// TIA Portal V17 export
// export: Created 2025-06-26T07:49:35.4692747Z, ExportSetting WithDefaults, DisplayName Totally Integrated Automation Portal, DisplayVersion V17 Update 8, DisplayName TIA Portal Openness, DisplayVersion V17 Update 8, DisplayName TIA Portal Version Control Interface, DisplayVersion V17, DisplayName STEP 7 Professional, DisplayVersion V17 Update 8, DisplayName STEP 7 Safety, DisplayVersion V17 Update 6, DisplayName WinCC Advanced, DisplayVersion V17 Update 8
DATA_BLOCK "DB_StaticData"   // DB32
{ S7_Optimized_Access := 'TRUE' }
AUTHOR : AZ
VERSION : 0.1
// stored: AutoNumber true, DBAccessibleFromOPCUA true, DBAccessibleFromWebserver true, InstanceOfName StaticData-STRUCT, InstanceOfType UDT, IsOnlyStoredInLoadMemory true, IsWriteProtectedInAS false
"StaticData-STRUCT"
   // VAR
   //    Fluids { ExternalAccessible := 'False'; ExternalVisible := 'False'; ExternalWritable := 'False'; S7_SetPoint := 'True'} : Array[1..4] of "FluidData-STRUCT";
   //    CompressorTypes { ExternalAccessible := 'False'; ExternalVisible := 'False'; ExternalWritable := 'False'; S7_SetPoint := 'True'} : Array[1..4] of "CompressorData-STRUCT";
   //    SystemTypes { ExternalAccessible := 'False'; ExternalVisible := 'False'; ExternalWritable := 'False'; S7_SetPoint := 'True'} : Array[1..6] of "SystemData-STRUCT";
   // END_VAR
BEGIN
   Fluids[1]."Name" := 'R515B';
   Fluids[2]."Name" := 'R1233zdE';
   Fluids[1].FluidTypeNumber := 1;
   Fluids[2].FluidTypeNumber := 2;
   Fluids[3].FluidTypeNumber := 3;
   Fluids[4].FluidTypeNumber := 4;
   Fluids[1].SaturationCurve_Temperature_C[0] := -43.0;
   Fluids[1].SaturationCurve_Temperature_C[1] := -39.15;
   Fluids[1].SaturationCurve_Temperature_C[2] := -35.31;
   Fluids[1].SaturationCurve_Temperature_C[3] := -31.46;
   Fluids[1].SaturationCurve_Temperature_C[4] := -27.62;
   Fluids[1].SaturationCurve_Temperature_C[5] := -23.77;
   Fluids[1].SaturationCurve_Temperature_C[6] := -19.92;
   Fluids[1].SaturationCurve_Temperature_C[7] := -16.08;
   Fluids[1].SaturationCurve_Temperature_C[8] := -12.23;
   Fluids[1].SaturationCurve_Temperature_C[9] := -8.38;
   Fluids[1].SaturationCurve_Temperature_C[10] := -4.54;
   Fluids[1].SaturationCurve_Temperature_C[11] := -0.69;
   Fluids[1].SaturationCurve_Temperature_C[12] := 3.15;
   Fluids[1].SaturationCurve_Temperature_C[13] := 7.0;
   Fluids[1].SaturationCurve_Temperature_C[14] := 10.85;
   Fluids[1].SaturationCurve_Temperature_C[15] := 14.69;
   Fluids[1].SaturationCurve_Temperature_C[16] := 18.54;
   Fluids[1].SaturationCurve_Temperature_C[17] := 22.38;
   Fluids[1].SaturationCurve_Temperature_C[18] := 26.23;
   Fluids[1].SaturationCurve_Temperature_C[19] := 30.08;
   Fluids[1].SaturationCurve_Temperature_C[20] := 33.92;
   Fluids[1].SaturationCurve_Temperature_C[21] := 37.77;
   Fluids[1].SaturationCurve_Temperature_C[22] := 41.62;
   Fluids[1].SaturationCurve_Temperature_C[23] := 45.46;
   Fluids[1].SaturationCurve_Temperature_C[24] := 49.31;
   Fluids[1].SaturationCurve_Temperature_C[25] := 53.15;
   Fluids[1].SaturationCurve_Temperature_C[26] := 57.0;
   Fluids[1].SaturationCurve_Temperature_C[27] := 60.85;
   Fluids[1].SaturationCurve_Temperature_C[28] := 64.69;
   Fluids[1].SaturationCurve_Temperature_C[29] := 68.54;
   Fluids[1].SaturationCurve_Temperature_C[30] := 72.38;
   Fluids[1].SaturationCurve_Temperature_C[31] := 76.23;
   Fluids[1].SaturationCurve_Temperature_C[32] := 80.08;
   Fluids[1].SaturationCurve_Temperature_C[33] := 83.92;
   Fluids[1].SaturationCurve_Temperature_C[34] := 87.77;
   Fluids[1].SaturationCurve_Temperature_C[35] := 91.62;
   Fluids[1].SaturationCurve_Temperature_C[36] := 95.46;
   Fluids[1].SaturationCurve_Temperature_C[37] := 99.31;
   Fluids[1].SaturationCurve_Temperature_C[38] := 103.15;
   Fluids[1].SaturationCurve_Temperature_C[39] := 107.0;
   Fluids[1].SaturationCurve_Temperature_C[40] := 107.73;
   Fluids[2].SaturationCurve_Temperature_C[0] := -10.0;
   Fluids[2].SaturationCurve_Temperature_C[1] := -5.4872;
   Fluids[2].SaturationCurve_Temperature_C[2] := -0.9744;
   Fluids[2].SaturationCurve_Temperature_C[3] := 3.5385;
   Fluids[2].SaturationCurve_Temperature_C[4] := 8.0513;
   Fluids[2].SaturationCurve_Temperature_C[5] := 12.5641;
   Fluids[2].SaturationCurve_Temperature_C[6] := 17.0769;
   Fluids[2].SaturationCurve_Temperature_C[7] := 21.5897;
   Fluids[2].SaturationCurve_Temperature_C[8] := 26.1026;
   Fluids[2].SaturationCurve_Temperature_C[9] := 30.6154;
   Fluids[2].SaturationCurve_Temperature_C[10] := 35.1282;
   Fluids[2].SaturationCurve_Temperature_C[11] := 39.641;
   Fluids[2].SaturationCurve_Temperature_C[12] := 44.1538;
   Fluids[2].SaturationCurve_Temperature_C[13] := 48.6667;
   Fluids[2].SaturationCurve_Temperature_C[14] := 53.1795;
   Fluids[2].SaturationCurve_Temperature_C[15] := 57.6923;
   Fluids[2].SaturationCurve_Temperature_C[16] := 62.2051;
   Fluids[2].SaturationCurve_Temperature_C[17] := 66.7179;
   Fluids[2].SaturationCurve_Temperature_C[18] := 71.2308;
   Fluids[2].SaturationCurve_Temperature_C[19] := 75.7436;
   Fluids[2].SaturationCurve_Temperature_C[20] := 80.2564;
   Fluids[2].SaturationCurve_Temperature_C[21] := 84.7692;
   Fluids[2].SaturationCurve_Temperature_C[22] := 89.2821;
   Fluids[2].SaturationCurve_Temperature_C[23] := 93.7949;
   Fluids[2].SaturationCurve_Temperature_C[24] := 98.3077;
   Fluids[2].SaturationCurve_Temperature_C[25] := 102.8205;
   Fluids[2].SaturationCurve_Temperature_C[26] := 107.3333;
   Fluids[2].SaturationCurve_Temperature_C[27] := 111.8462;
   Fluids[2].SaturationCurve_Temperature_C[28] := 116.359;
   Fluids[2].SaturationCurve_Temperature_C[29] := 120.8718;
   Fluids[2].SaturationCurve_Temperature_C[30] := 125.3846;
   Fluids[2].SaturationCurve_Temperature_C[31] := 129.8974;
   Fluids[2].SaturationCurve_Temperature_C[32] := 134.4103;
   Fluids[2].SaturationCurve_Temperature_C[33] := 138.9231;
   Fluids[2].SaturationCurve_Temperature_C[34] := 143.4359;
   Fluids[2].SaturationCurve_Temperature_C[35] := 147.9487;
   Fluids[2].SaturationCurve_Temperature_C[36] := 152.4615;
   Fluids[2].SaturationCurve_Temperature_C[37] := 156.9744;
   Fluids[2].SaturationCurve_Temperature_C[38] := 161.4872;
   Fluids[2].SaturationCurve_Temperature_C[39] := 166.0;
   Fluids[2].SaturationCurve_Temperature_C[40] := 172.9092;
   Fluids[1].SaturationCurve_Pressure_kPa[0] := 30.9;
   Fluids[1].SaturationCurve_Pressure_kPa[1] := 38.1;
   Fluids[1].SaturationCurve_Pressure_kPa[2] := 46.5;
   Fluids[1].SaturationCurve_Pressure_kPa[3] := 56.4;
   Fluids[1].SaturationCurve_Pressure_kPa[4] := 67.9;
   Fluids[1].SaturationCurve_Pressure_kPa[5] := 81.1;
   Fluids[1].SaturationCurve_Pressure_kPa[6] := 96.4;
   Fluids[1].SaturationCurve_Pressure_kPa[7] := 113.8;
   Fluids[1].SaturationCurve_Pressure_kPa[8] := 133.6;
   Fluids[1].SaturationCurve_Pressure_kPa[9] := 156.0;
   Fluids[1].SaturationCurve_Pressure_kPa[10] := 181.2;
   Fluids[1].SaturationCurve_Pressure_kPa[11] := 209.5;
   Fluids[1].SaturationCurve_Pressure_kPa[12] := 241.0;
   Fluids[1].SaturationCurve_Pressure_kPa[13] := 276.1;
   Fluids[1].SaturationCurve_Pressure_kPa[14] := 315.0;
   Fluids[1].SaturationCurve_Pressure_kPa[15] := 358.0;
   Fluids[1].SaturationCurve_Pressure_kPa[16] := 405.2;
   Fluids[1].SaturationCurve_Pressure_kPa[17] := 457.1;
   Fluids[1].SaturationCurve_Pressure_kPa[18] := 513.8;
   Fluids[1].SaturationCurve_Pressure_kPa[19] := 575.8;
   Fluids[1].SaturationCurve_Pressure_kPa[20] := 643.2;
   Fluids[1].SaturationCurve_Pressure_kPa[21] := 716.3;
   Fluids[1].SaturationCurve_Pressure_kPa[22] := 795.6;
   Fluids[1].SaturationCurve_Pressure_kPa[23] := 881.2;
   Fluids[1].SaturationCurve_Pressure_kPa[24] := 973.6;
   Fluids[1].SaturationCurve_Pressure_kPa[25] := 1073.1;
   Fluids[1].SaturationCurve_Pressure_kPa[26] := 1180.0;
   Fluids[1].SaturationCurve_Pressure_kPa[27] := 1294.8;
   Fluids[1].SaturationCurve_Pressure_kPa[28] := 1417.7;
   Fluids[1].SaturationCurve_Pressure_kPa[29] := 1549.2;
   Fluids[1].SaturationCurve_Pressure_kPa[30] := 1689.7;
   Fluids[1].SaturationCurve_Pressure_kPa[31] := 1839.6;
   Fluids[1].SaturationCurve_Pressure_kPa[32] := 1999.6;
   Fluids[1].SaturationCurve_Pressure_kPa[33] := 2169.9;
   Fluids[1].SaturationCurve_Pressure_kPa[34] := 2351.3;
   Fluids[1].SaturationCurve_Pressure_kPa[35] := 2544.5;
   Fluids[1].SaturationCurve_Pressure_kPa[36] := 2750.1;
   Fluids[1].SaturationCurve_Pressure_kPa[37] := 2969.2;
   Fluids[1].SaturationCurve_Pressure_kPa[38] := 3202.9;
   Fluids[1].SaturationCurve_Pressure_kPa[39] := 3453.4;
   Fluids[1].SaturationCurve_Pressure_kPa[40] := 3501.0;
   Fluids[2].SaturationCurve_Pressure_kPa[0] := 30.3567;
   Fluids[2].SaturationCurve_Pressure_kPa[1] := 37.5596;
   Fluids[2].SaturationCurve_Pressure_kPa[2] := 46.0817;
   Fluids[2].SaturationCurve_Pressure_kPa[3] := 56.0903;
   Fluids[2].SaturationCurve_Pressure_kPa[4] := 67.7633;
   Fluids[2].SaturationCurve_Pressure_kPa[5] := 81.2888;
   Fluids[2].SaturationCurve_Pressure_kPa[6] := 96.865;
   Fluids[2].SaturationCurve_Pressure_kPa[7] := 114.6997;
   Fluids[2].SaturationCurve_Pressure_kPa[8] := 135.0095;
   Fluids[2].SaturationCurve_Pressure_kPa[9] := 158.0203;
   Fluids[2].SaturationCurve_Pressure_kPa[10] := 183.9659;
   Fluids[2].SaturationCurve_Pressure_kPa[11] := 213.0886;
   Fluids[2].SaturationCurve_Pressure_kPa[12] := 245.6381;
   Fluids[2].SaturationCurve_Pressure_kPa[13] := 281.8717;
   Fluids[2].SaturationCurve_Pressure_kPa[14] := 322.0539;
   Fluids[2].SaturationCurve_Pressure_kPa[15] := 366.4563;
   Fluids[2].SaturationCurve_Pressure_kPa[16] := 415.3576;
   Fluids[2].SaturationCurve_Pressure_kPa[17] := 469.0435;
   Fluids[2].SaturationCurve_Pressure_kPa[18] := 527.8071;
   Fluids[2].SaturationCurve_Pressure_kPa[19] := 591.9489;
   Fluids[2].SaturationCurve_Pressure_kPa[20] := 661.7775;
   Fluids[2].SaturationCurve_Pressure_kPa[21] := 737.6098;
   Fluids[2].SaturationCurve_Pressure_kPa[22] := 819.7723;
   Fluids[2].SaturationCurve_Pressure_kPa[23] := 908.6015;
   Fluids[2].SaturationCurve_Pressure_kPa[24] := 1004.446;
   Fluids[2].SaturationCurve_Pressure_kPa[25] := 1107.666;
   Fluids[2].SaturationCurve_Pressure_kPa[26] := 1218.639;
   Fluids[2].SaturationCurve_Pressure_kPa[27] := 1337.757;
   Fluids[2].SaturationCurve_Pressure_kPa[28] := 1465.436;
   Fluids[2].SaturationCurve_Pressure_kPa[29] := 1602.111;
   Fluids[2].SaturationCurve_Pressure_kPa[30] := 1748.251;
   Fluids[2].SaturationCurve_Pressure_kPa[31] := 1904.356;
   Fluids[2].SaturationCurve_Pressure_kPa[32] := 2070.969;
   Fluids[2].SaturationCurve_Pressure_kPa[33] := 2248.688;
   Fluids[2].SaturationCurve_Pressure_kPa[34] := 2438.177;
   Fluids[2].SaturationCurve_Pressure_kPa[35] := 2640.193;
   Fluids[2].SaturationCurve_Pressure_kPa[36] := 2855.623;
   Fluids[2].SaturationCurve_Pressure_kPa[37] := 3085.555;
   Fluids[2].SaturationCurve_Pressure_kPa[38] := 3331.466;
   Fluids[2].SaturationCurve_Pressure_kPa[39] := 3595.998;
   Fluids[2].SaturationCurve_Pressure_kPa[40] := 4001.0;
   Fluids[1].DensityCurve_Pressure_kPa[0] := 50.0;
   Fluids[1].DensityCurve_Pressure_kPa[1] := 100.0;
   Fluids[1].DensityCurve_Pressure_kPa[2] := 220.0;
   Fluids[1].DensityCurve_Pressure_kPa[3] := 390.0;
   Fluids[1].DensityCurve_Pressure_kPa[4] := 600.0;
   Fluids[1].DensityCurve_Pressure_kPa[5] := 850.0;
   Fluids[1].DensityCurve_Pressure_kPa[6] := 1200.0;
   Fluids[1].DensityCurve_Pressure_kPa[7] := 1500.0;
   Fluids[1].DensityCurve_Pressure_kPa[8] := 1900.0;
   Fluids[1].DensityCurve_Pressure_kPa[9] := 2400.0;
   Fluids[1].DensityCurve_Pressure_kPa[10] := 2900.0;
   Fluids[1].DensityCurve_Pressure_kPa[11] := 3400.0;
   Fluids[1].DensityCurve_Pressure_kPa[12] := 4000.0;
   Fluids[2].DensityCurve_Pressure_kPa[0] := 50.0;
   Fluids[2].DensityCurve_Pressure_kPa[1] := 74.7475;
   Fluids[2].DensityCurve_Pressure_kPa[2] := 173.05;
   Fluids[2].DensityCurve_Pressure_kPa[3] := 388.0866;
   Fluids[2].DensityCurve_Pressure_kPa[4] := 746.4811;
   Fluids[2].DensityCurve_Pressure_kPa[5] := 1244.251;
   Fluids[2].DensityCurve_Pressure_kPa[6] := 1836.598;
   Fluids[2].DensityCurve_Pressure_kPa[7] := 2441.284;
   Fluids[2].DensityCurve_Pressure_kPa[8] := 2962.33;
   Fluids[2].DensityCurve_Pressure_kPa[9] := 3328.69;
   Fluids[2].DensityCurve_Pressure_kPa[10] := 3526.57;
   Fluids[2].DensityCurve_Pressure_kPa[11] := 3613.637;
   Fluids[2].DensityCurve_Pressure_kPa[12] := 4001.0;
   Fluids[1].DensityCurveLiquide_Densety_kg_m3[0] := 1354.6;
   Fluids[1].DensityCurveLiquide_Densety_kg_m3[1] := 1314.3;
   Fluids[1].DensityCurveLiquide_Densety_kg_m3[2] := 1257.6;
   Fluids[1].DensityCurveLiquide_Densety_kg_m3[3] := 1206.1;
   Fluids[1].DensityCurveLiquide_Densety_kg_m3[4] := 1158.8;
   Fluids[1].DensityCurveLiquide_Densety_kg_m3[5] := 1113.0;
   Fluids[1].DensityCurveLiquide_Densety_kg_m3[6] := 1057.8;
   Fluids[1].DensityCurveLiquide_Densety_kg_m3[7] := 1014.5;
   Fluids[1].DensityCurveLiquide_Densety_kg_m3[8] := 958.8;
   Fluids[1].DensityCurveLiquide_Densety_kg_m3[9] := 887.4;
   Fluids[1].DensityCurveLiquide_Densety_kg_m3[10] := 805.7;
   Fluids[1].DensityCurveLiquide_Densety_kg_m3[11] := 685.3;
   Fluids[1].DensityCurveLiquide_Densety_kg_m3[12] := 761.3;
   Fluids[2].DensityCurveLiquide_Densety_kg_m3[0] := 1319.278;
   Fluids[2].DensityCurveLiquide_Densety_kg_m3[1] := 1297.254;
   Fluids[2].DensityCurveLiquide_Densety_kg_m3[2] := 1242.459;
   Fluids[2].DensityCurveLiquide_Densety_kg_m3[3] := 1173.489;
   Fluids[2].DensityCurveLiquide_Densety_kg_m3[4] := 1098.545;
   Fluids[2].DensityCurveLiquide_Densety_kg_m3[5] := 1019.4;
   Fluids[2].DensityCurveLiquide_Densety_kg_m3[6] := 936.68;
   Fluids[2].DensityCurveLiquide_Densety_kg_m3[7] := 851.4562;
   Fluids[2].DensityCurveLiquide_Densety_kg_m3[8] := 765.7374;
   Fluids[2].DensityCurveLiquide_Densety_kg_m3[9] := 682.3312;
   Fluids[2].DensityCurveLiquide_Densety_kg_m3[10] := 605.4245;
   Fluids[2].DensityCurveLiquide_Densety_kg_m3[11] := 523.5075;
   Fluids[2].DensityCurveLiquide_Densety_kg_m3[12] := 455.9911;
   Fluids[1].DensityCurveVapor_Densety_kg_m3[0] := 3.03;
   Fluids[1].DensityCurveVapor_Densety_kg_m3[1] := 5.8;
   Fluids[1].DensityCurveVapor_Densety_kg_m3[2] := 12.25;
   Fluids[1].DensityCurveVapor_Densety_kg_m3[3] := 21.3;
   Fluids[1].DensityCurveVapor_Densety_kg_m3[4] := 32.65;
   Fluids[1].DensityCurveVapor_Densety_kg_m3[5] := 46.66;
   Fluids[1].DensityCurveVapor_Densety_kg_m3[6] := 67.55;
   Fluids[1].DensityCurveVapor_Densety_kg_m3[7] := 87.0;
   Fluids[1].DensityCurveVapor_Densety_kg_m3[8] := 115.92;
   Fluids[1].DensityCurveVapor_Densety_kg_m3[9] := 159.17;
   Fluids[1].DensityCurveVapor_Densety_kg_m3[10] := 216.59;
   Fluids[1].DensityCurveVapor_Densety_kg_m3[11] := 315.0;
   Fluids[1].DensityCurveVapor_Densety_kg_m3[12] := 761.33;
   Fluids[2].DensityCurveVapor_Densety_kg_m3[0] := 2.9405;
   Fluids[2].DensityCurveVapor_Densety_kg_m3[1] := 4.2862;
   Fluids[2].DensityCurveVapor_Densety_kg_m3[2] := 9.4624;
   Fluids[2].DensityCurveVapor_Densety_kg_m3[3] := 20.5809;
   Fluids[2].DensityCurveVapor_Densety_kg_m3[4] := 39.5976;
   Fluids[2].DensityCurveVapor_Densety_kg_m3[5] := 68.316;
   Fluids[2].DensityCurveVapor_Densety_kg_m3[6] := 108.1358;
   Fluids[2].DensityCurveVapor_Densety_kg_m3[7] := 159.5525;
   Fluids[2].DensityCurveVapor_Densety_kg_m3[8] := 221.352;
   Fluids[2].DensityCurveVapor_Densety_kg_m3[9] := 289.9457;
   Fluids[2].DensityCurveVapor_Densety_kg_m3[10] := 359.0497;
   Fluids[2].DensityCurveVapor_Densety_kg_m3[11] := 437.3655;
   Fluids[2].DensityCurveVapor_Densety_kg_m3[12] := 455.9911;
   Fluids[1].DensityCurveVapor_SuperheatCorrection_a := 1.3561E-07;
   Fluids[2].DensityCurveVapor_SuperheatCorrection_a := 0.0;
   Fluids[1].DensityCurveVapor_SuperheatCorrection_b := 0.00019589;
   Fluids[2].DensityCurveVapor_SuperheatCorrection_b := 0.0002;
   Fluids[1].EnthalpyMap_Superheat_C[0] := -20.0;
   Fluids[1].EnthalpyMap_Superheat_C[1] := -6.0;
   Fluids[1].EnthalpyMap_Superheat_C[2] := -2.0;
   Fluids[1].EnthalpyMap_Superheat_C[3] := -0.01;
   Fluids[1].EnthalpyMap_Superheat_C[4] := 0.01;
   Fluids[1].EnthalpyMap_Superheat_C[5] := 2.0;
   Fluids[1].EnthalpyMap_Superheat_C[6] := 6.0;
   Fluids[1].EnthalpyMap_Superheat_C[7] := 18.0;
   Fluids[1].EnthalpyMap_Superheat_C[8] := 40.0;
   Fluids[2].EnthalpyMap_Superheat_C[0] := -20.0;
   Fluids[2].EnthalpyMap_Superheat_C[1] := -6.0;
   Fluids[2].EnthalpyMap_Superheat_C[2] := -2.0;
   Fluids[2].EnthalpyMap_Superheat_C[3] := -0.01;
   Fluids[2].EnthalpyMap_Superheat_C[4] := 0.01;
   Fluids[2].EnthalpyMap_Superheat_C[5] := 2.0;
   Fluids[2].EnthalpyMap_Superheat_C[6] := 6.0;
   Fluids[2].EnthalpyMap_Superheat_C[7] := 18.0;
   Fluids[2].EnthalpyMap_Superheat_C[8] := 40.0;
   Fluids[1].EnthalpyMap_Pressure_kPa[0] := 100.0;
   Fluids[1].EnthalpyMap_Pressure_kPa[1] := 220.0;
   Fluids[1].EnthalpyMap_Pressure_kPa[2] := 390.0;
   Fluids[1].EnthalpyMap_Pressure_kPa[3] := 600.0;
   Fluids[1].EnthalpyMap_Pressure_kPa[4] := 850.0;
   Fluids[1].EnthalpyMap_Pressure_kPa[5] := 1200.0;
   Fluids[1].EnthalpyMap_Pressure_kPa[6] := 1500.0;
   Fluids[1].EnthalpyMap_Pressure_kPa[7] := 1900.0;
   Fluids[1].EnthalpyMap_Pressure_kPa[8] := 2400.0;
   Fluids[1].EnthalpyMap_Pressure_kPa[9] := 2900.0;
   Fluids[1].EnthalpyMap_Pressure_kPa[10] := 3400.0;
   Fluids[1].EnthalpyMap_Pressure_kPa[11] := 4000.0;
   Fluids[2].EnthalpyMap_Pressure_kPa[0] := 100.0;
   Fluids[2].EnthalpyMap_Pressure_kPa[1] := 127.0833;
   Fluids[2].EnthalpyMap_Pressure_kPa[2] := 234.6644;
   Fluids[2].EnthalpyMap_Pressure_kPa[3] := 469.9978;
   Fluids[2].EnthalpyMap_Pressure_kPa[4] := 862.2203;
   Fluids[2].EnthalpyMap_Pressure_kPa[5] := 1406.974;
   Fluids[2].EnthalpyMap_Pressure_kPa[6] := 2055.23;
   Fluids[2].EnthalpyMap_Pressure_kPa[7] := 2716.992;
   Fluids[2].EnthalpyMap_Pressure_kPa[8] := 3287.218;
   Fluids[2].EnthalpyMap_Pressure_kPa[9] := 3688.158;
   Fluids[2].EnthalpyMap_Pressure_kPa[10] := 3904.715;
   Fluids[2].EnthalpyMap_Pressure_kPa[11] := 4000.0;
   Fluids[1].EnthalpyMap_Enthalpy_kJ_kg[0,0] := 150.5;
   Fluids[1].EnthalpyMap_Enthalpy_kJ_kg[0,1] := 167.9;
   Fluids[1].EnthalpyMap_Enthalpy_kJ_kg[0,2] := 173.0;
   Fluids[1].EnthalpyMap_Enthalpy_kJ_kg[0,3] := 175.5;
   Fluids[1].EnthalpyMap_Enthalpy_kJ_kg[0,4] := 271.8;
   Fluids[1].EnthalpyMap_Enthalpy_kJ_kg[0,5] := 367.3;
   Fluids[1].EnthalpyMap_Enthalpy_kJ_kg[0,6] := 370.6;
   Fluids[1].EnthalpyMap_Enthalpy_kJ_kg[0,7] := 380.6;
   Fluids[1].EnthalpyMap_Enthalpy_kJ_kg[0,8] := 399.6;
   Fluids[1].EnthalpyMap_Enthalpy_kJ_kg[1,0] := 175.2;
   Fluids[1].EnthalpyMap_Enthalpy_kJ_kg[1,1] := 193.0;
   Fluids[1].EnthalpyMap_Enthalpy_kJ_kg[1,2] := 198.2;
   Fluids[1].EnthalpyMap_Enthalpy_kJ_kg[1,3] := 200.8;
   Fluids[1].EnthalpyMap_Enthalpy_kJ_kg[1,4] := 297.6;
   Fluids[1].EnthalpyMap_Enthalpy_kJ_kg[1,5] := 381.1;
   Fluids[1].EnthalpyMap_Enthalpy_kJ_kg[1,6] := 384.6;
   Fluids[1].EnthalpyMap_Enthalpy_kJ_kg[1,7] := 395.3;
   Fluids[1].EnthalpyMap_Enthalpy_kJ_kg[1,8] := 415.2;
   Fluids[1].EnthalpyMap_Enthalpy_kJ_kg[2,0] := 196.6;
   Fluids[1].EnthalpyMap_Enthalpy_kJ_kg[2,1] := 214.9;
   Fluids[1].EnthalpyMap_Enthalpy_kJ_kg[2,2] := 220.2;
   Fluids[1].EnthalpyMap_Enthalpy_kJ_kg[2,3] := 222.9;
   Fluids[1].EnthalpyMap_Enthalpy_kJ_kg[2,4] := 318.7;
   Fluids[1].EnthalpyMap_Enthalpy_kJ_kg[2,5] := 392.3;
   Fluids[1].EnthalpyMap_Enthalpy_kJ_kg[2,6] := 396.1;
   Fluids[1].EnthalpyMap_Enthalpy_kJ_kg[2,7] := 407.4;
   Fluids[1].EnthalpyMap_Enthalpy_kJ_kg[2,8] := 428.3;
   Fluids[1].EnthalpyMap_Enthalpy_kJ_kg[3,0] := 215.2;
   Fluids[1].EnthalpyMap_Enthalpy_kJ_kg[3,1] := 234.0;
   Fluids[1].EnthalpyMap_Enthalpy_kJ_kg[3,2] := 239.5;
   Fluids[1].EnthalpyMap_Enthalpy_kJ_kg[3,3] := 242.3;
   Fluids[1].EnthalpyMap_Enthalpy_kJ_kg[3,4] := 336.5;
   Fluids[1].EnthalpyMap_Enthalpy_kJ_kg[3,5] := 401.4;
   Fluids[1].EnthalpyMap_Enthalpy_kJ_kg[3,6] := 405.3;
   Fluids[1].EnthalpyMap_Enthalpy_kJ_kg[3,7] := 417.3;
   Fluids[1].EnthalpyMap_Enthalpy_kJ_kg[3,8] := 439.2;
   Fluids[1].EnthalpyMap_Enthalpy_kJ_kg[4,0] := 232.1;
   Fluids[1].EnthalpyMap_Enthalpy_kJ_kg[4,1] := 251.5;
   Fluids[1].EnthalpyMap_Enthalpy_kJ_kg[4,2] := 257.2;
   Fluids[1].EnthalpyMap_Enthalpy_kJ_kg[4,3] := 260.1;
   Fluids[1].EnthalpyMap_Enthalpy_kJ_kg[4,4] := 352.6;
   Fluids[1].EnthalpyMap_Enthalpy_kJ_kg[4,5] := 408.9;
   Fluids[1].EnthalpyMap_Enthalpy_kJ_kg[4,6] := 413.1;
   Fluids[1].EnthalpyMap_Enthalpy_kJ_kg[4,7] := 425.7;
   Fluids[1].EnthalpyMap_Enthalpy_kJ_kg[4,8] := 448.6;
   Fluids[1].EnthalpyMap_Enthalpy_kJ_kg[5,0] := 251.0;
   Fluids[1].EnthalpyMap_Enthalpy_kJ_kg[5,1] := 271.1;
   Fluids[1].EnthalpyMap_Enthalpy_kJ_kg[5,2] := 277.1;
   Fluids[1].EnthalpyMap_Enthalpy_kJ_kg[5,3] := 280.1;
   Fluids[1].EnthalpyMap_Enthalpy_kJ_kg[5,4] := 370.8;
   Fluids[1].EnthalpyMap_Enthalpy_kJ_kg[5,5] := 416.2;
   Fluids[1].EnthalpyMap_Enthalpy_kJ_kg[5,6] := 420.8;
   Fluids[1].EnthalpyMap_Enthalpy_kJ_kg[5,7] := 434.3;
   Fluids[1].EnthalpyMap_Enthalpy_kJ_kg[5,8] := 458.5;
   Fluids[1].EnthalpyMap_Enthalpy_kJ_kg[6,0] := 264.4;
   Fluids[1].EnthalpyMap_Enthalpy_kJ_kg[6,1] := 285.3;
   Fluids[1].EnthalpyMap_Enthalpy_kJ_kg[6,2] := 291.5;
   Fluids[1].EnthalpyMap_Enthalpy_kJ_kg[6,3] := 294.7;
   Fluids[1].EnthalpyMap_Enthalpy_kJ_kg[6,4] := 384.4;
   Fluids[1].EnthalpyMap_Enthalpy_kJ_kg[6,5] := 420.5;
   Fluids[1].EnthalpyMap_Enthalpy_kJ_kg[6,6] := 425.5;
   Fluids[1].EnthalpyMap_Enthalpy_kJ_kg[6,7] := 439.9;
   Fluids[1].EnthalpyMap_Enthalpy_kJ_kg[6,8] := 465.0;
   Fluids[1].EnthalpyMap_Enthalpy_kJ_kg[7,0] := 279.9;
   Fluids[1].EnthalpyMap_Enthalpy_kJ_kg[7,1] := 301.7;
   Fluids[1].EnthalpyMap_Enthalpy_kJ_kg[7,2] := 308.4;
   Fluids[1].EnthalpyMap_Enthalpy_kJ_kg[7,3] := 311.8;
   Fluids[1].EnthalpyMap_Enthalpy_kJ_kg[7,4] := 401.2;
   Fluids[1].EnthalpyMap_Enthalpy_kJ_kg[7,5] := 424.5;
   Fluids[1].EnthalpyMap_Enthalpy_kJ_kg[7,6] := 430.0;
   Fluids[1].EnthalpyMap_Enthalpy_kJ_kg[7,7] := 445.6;
   Fluids[1].EnthalpyMap_Enthalpy_kJ_kg[7,8] := 472.1;
   Fluids[1].EnthalpyMap_Enthalpy_kJ_kg[8,0] := 296.6;
   Fluids[1].EnthalpyMap_Enthalpy_kJ_kg[8,1] := 319.8;
   Fluids[1].EnthalpyMap_Enthalpy_kJ_kg[8,2] := 327.2;
   Fluids[1].EnthalpyMap_Enthalpy_kJ_kg[8,3] := 331.1;
   Fluids[1].EnthalpyMap_Enthalpy_kJ_kg[8,4] := 422.0;
   Fluids[1].EnthalpyMap_Enthalpy_kJ_kg[8,5] := 427.0;
   Fluids[1].EnthalpyMap_Enthalpy_kJ_kg[8,6] := 433.5;
   Fluids[1].EnthalpyMap_Enthalpy_kJ_kg[8,7] := 450.9;
   Fluids[1].EnthalpyMap_Enthalpy_kJ_kg[8,8] := 479.1;
   Fluids[1].EnthalpyMap_Enthalpy_kJ_kg[9,0] := 311.2;
   Fluids[1].EnthalpyMap_Enthalpy_kJ_kg[9,1] := 336.2;
   Fluids[1].EnthalpyMap_Enthalpy_kJ_kg[9,2] := 344.7;
   Fluids[1].EnthalpyMap_Enthalpy_kJ_kg[9,3] := 349.5;
   Fluids[1].EnthalpyMap_Enthalpy_kJ_kg[9,4] := 421.8;
   Fluids[1].EnthalpyMap_Enthalpy_kJ_kg[9,5] := 426.9;
   Fluids[1].EnthalpyMap_Enthalpy_kJ_kg[9,6] := 435.1;
   Fluids[1].EnthalpyMap_Enthalpy_kJ_kg[9,7] := 454.7;
   Fluids[1].EnthalpyMap_Enthalpy_kJ_kg[9,8] := 484.7;
   Fluids[1].EnthalpyMap_Enthalpy_kJ_kg[10,0] := 324.2;
   Fluids[1].EnthalpyMap_Enthalpy_kJ_kg[10,1] := 351.3;
   Fluids[1].EnthalpyMap_Enthalpy_kJ_kg[10,2] := 361.9;
   Fluids[1].EnthalpyMap_Enthalpy_kJ_kg[10,3] := 370.2;
   Fluids[1].EnthalpyMap_Enthalpy_kJ_kg[10,4] := 413.6;
   Fluids[1].EnthalpyMap_Enthalpy_kJ_kg[10,5] := 423.8;
   Fluids[1].EnthalpyMap_Enthalpy_kJ_kg[10,6] := 434.9;
   Fluids[1].EnthalpyMap_Enthalpy_kJ_kg[10,7] := 457.3;
   Fluids[1].EnthalpyMap_Enthalpy_kJ_kg[10,8] := 489.2;
   Fluids[1].EnthalpyMap_Enthalpy_kJ_kg[11,0] := 339.4;
   Fluids[1].EnthalpyMap_Enthalpy_kJ_kg[11,1] := 370.1;
   Fluids[1].EnthalpyMap_Enthalpy_kJ_kg[11,2] := 387.3;
   Fluids[1].EnthalpyMap_Enthalpy_kJ_kg[11,3] := 407.7;
   Fluids[1].EnthalpyMap_Enthalpy_kJ_kg[11,4] := 407.9;
   Fluids[1].EnthalpyMap_Enthalpy_kJ_kg[11,5] := 421.3;
   Fluids[1].EnthalpyMap_Enthalpy_kJ_kg[11,6] := 435.4;
   Fluids[1].EnthalpyMap_Enthalpy_kJ_kg[11,7] := 460.7;
   Fluids[1].EnthalpyMap_Enthalpy_kJ_kg[11,8] := 494.6;
   Fluids[2].EnthalpyMap_Enthalpy_kJ_kg[0,0] := 197.5698;
   Fluids[2].EnthalpyMap_Enthalpy_kJ_kg[0,1] := 214.1515;
   Fluids[2].EnthalpyMap_Enthalpy_kJ_kg[0,2] := 218.9438;
   Fluids[2].EnthalpyMap_Enthalpy_kJ_kg[0,3] := 221.3373;
   Fluids[2].EnthalpyMap_Enthalpy_kJ_kg[0,4] := 416.1527;
   Fluids[2].EnthalpyMap_Enthalpy_kJ_kg[0,5] := 417.767;
   Fluids[2].EnthalpyMap_Enthalpy_kJ_kg[0,6] := 421.028;
   Fluids[2].EnthalpyMap_Enthalpy_kJ_kg[0,7] := 430.9391;
   Fluids[2].EnthalpyMap_Enthalpy_kJ_kg[0,8] := 449.5907;
   Fluids[2].EnthalpyMap_Enthalpy_kJ_kg[1,0] := 205.2355;
   Fluids[2].EnthalpyMap_Enthalpy_kJ_kg[1,1] := 221.9542;
   Fluids[2].EnthalpyMap_Enthalpy_kJ_kg[1,2] := 226.7875;
   Fluids[2].EnthalpyMap_Enthalpy_kJ_kg[1,3] := 229.2018;
   Fluids[2].EnthalpyMap_Enthalpy_kJ_kg[1,4] := 420.6821;
   Fluids[2].EnthalpyMap_Enthalpy_kJ_kg[1,5] := 422.3276;
   Fluids[2].EnthalpyMap_Enthalpy_kJ_kg[1,6] := 425.6502;
   Fluids[2].EnthalpyMap_Enthalpy_kJ_kg[1,7] := 435.7365;
   Fluids[2].EnthalpyMap_Enthalpy_kJ_kg[1,8] := 454.6786;
   Fluids[2].EnthalpyMap_Enthalpy_kJ_kg[2,0] := 227.161;
   Fluids[2].EnthalpyMap_Enthalpy_kJ_kg[2,1] := 244.2909;
   Fluids[2].EnthalpyMap_Enthalpy_kJ_kg[2,2] := 249.2492;
   Fluids[2].EnthalpyMap_Enthalpy_kJ_kg[2,3] := 251.7272;
   Fluids[2].EnthalpyMap_Enthalpy_kJ_kg[2,4] := 433.2917;
   Fluids[2].EnthalpyMap_Enthalpy_kJ_kg[2,5] := 435.0327;
   Fluids[2].EnthalpyMap_Enthalpy_kJ_kg[2,6] := 438.5429;
   Fluids[2].EnthalpyMap_Enthalpy_kJ_kg[2,7] := 449.1592;
   Fluids[2].EnthalpyMap_Enthalpy_kJ_kg[2,8] := 468.9681;
   Fluids[2].EnthalpyMap_Enthalpy_kJ_kg[3,0] := 256.9384;
   Fluids[2].EnthalpyMap_Enthalpy_kJ_kg[3,1] := 274.7034;
   Fluids[2].EnthalpyMap_Enthalpy_kJ_kg[3,2] := 279.8614;
   Fluids[2].EnthalpyMap_Enthalpy_kJ_kg[3,3] := 282.4424;
   Fluids[2].EnthalpyMap_Enthalpy_kJ_kg[3,4] := 449.3674;
   Fluids[2].EnthalpyMap_Enthalpy_kJ_kg[3,5] := 451.2598;
   Fluids[2].EnthalpyMap_Enthalpy_kJ_kg[3,6] := 455.0643;
   Fluids[2].EnthalpyMap_Enthalpy_kJ_kg[3,7] := 466.4958;
   Fluids[2].EnthalpyMap_Enthalpy_kJ_kg[3,8] := 487.595;
   Fluids[2].EnthalpyMap_Enthalpy_kJ_kg[4,0] := 288.6115;
   Fluids[2].EnthalpyMap_Enthalpy_kJ_kg[4,1] := 307.2277;
   Fluids[2].EnthalpyMap_Enthalpy_kJ_kg[4,2] := 312.6681;
   Fluids[2].EnthalpyMap_Enthalpy_kJ_kg[4,3] := 315.398;
   Fluids[2].EnthalpyMap_Enthalpy_kJ_kg[4,4] := 464.6608;
   Fluids[2].EnthalpyMap_Enthalpy_kJ_kg[4,5] := 466.762;
   Fluids[2].EnthalpyMap_Enthalpy_kJ_kg[4,6] := 470.9658;
   Fluids[2].EnthalpyMap_Enthalpy_kJ_kg[4,7] := 483.4603;
   Fluids[2].EnthalpyMap_Enthalpy_kJ_kg[4,8] := 506.1447;
   Fluids[2].EnthalpyMap_Enthalpy_kJ_kg[5,0] := 319.2484;
   Fluids[2].EnthalpyMap_Enthalpy_kJ_kg[5,1] := 339.0134;
   Fluids[2].EnthalpyMap_Enthalpy_kJ_kg[5,2] := 344.8686;
   Fluids[2].EnthalpyMap_Enthalpy_kJ_kg[5,3] := 347.8254;
   Fluids[2].EnthalpyMap_Enthalpy_kJ_kg[5,4] := 476.8875;
   Fluids[2].EnthalpyMap_Enthalpy_kJ_kg[5,5] := 479.2968;
   Fluids[2].EnthalpyMap_Enthalpy_kJ_kg[5,6] := 484.0675;
   Fluids[2].EnthalpyMap_Enthalpy_kJ_kg[5,7] := 497.9603;
   Fluids[2].EnthalpyMap_Enthalpy_kJ_kg[5,8] := 522.524;
   Fluids[2].EnthalpyMap_Enthalpy_kJ_kg[6,0] := 346.9259;
   Fluids[2].EnthalpyMap_Enthalpy_kJ_kg[6,1] := 368.272;
   Fluids[2].EnthalpyMap_Enthalpy_kJ_kg[6,2] := 374.7868;
   Fluids[2].EnthalpyMap_Enthalpy_kJ_kg[6,3] := 378.132;
   Fluids[2].EnthalpyMap_Enthalpy_kJ_kg[6,4] := 484.4899;
   Fluids[2].EnthalpyMap_Enthalpy_kJ_kg[6,5] := 487.4372;
   Fluids[2].EnthalpyMap_Enthalpy_kJ_kg[6,6] := 493.119;
   Fluids[2].EnthalpyMap_Enthalpy_kJ_kg[6,7] := 508.9522;
   Fluids[2].EnthalpyMap_Enthalpy_kJ_kg[6,8] := 535.7144;
   Fluids[2].EnthalpyMap_Enthalpy_kJ_kg[7,0] := 369.9632;
   Fluids[2].EnthalpyMap_Enthalpy_kJ_kg[7,1] := 393.4236;
   Fluids[2].EnthalpyMap_Enthalpy_kJ_kg[7,2] := 401.0829;
   Fluids[2].EnthalpyMap_Enthalpy_kJ_kg[7,3] := 405.235;
   Fluids[2].EnthalpyMap_Enthalpy_kJ_kg[7,4] := 486.2374;
   Fluids[2].EnthalpyMap_Enthalpy_kJ_kg[7,5] := 490.3629;
   Fluids[2].EnthalpyMap_Enthalpy_kJ_kg[7,6] := 497.6848;
   Fluids[2].EnthalpyMap_Enthalpy_kJ_kg[7,7] := 516.2058;
   Fluids[2].EnthalpyMap_Enthalpy_kJ_kg[7,8] := 545.3667;
   Fluids[2].EnthalpyMap_Enthalpy_kJ_kg[8,0] := 387.0381;
   Fluids[2].EnthalpyMap_Enthalpy_kJ_kg[8,1] := 412.9451;
   Fluids[2].EnthalpyMap_Enthalpy_kJ_kg[8,2] := 422.6469;
   Fluids[2].EnthalpyMap_Enthalpy_kJ_kg[8,3] := 429.1883;
   Fluids[2].EnthalpyMap_Enthalpy_kJ_kg[8,4] := 480.7851;
   Fluids[2].EnthalpyMap_Enthalpy_kJ_kg[8,5] := 488.3624;
   Fluids[2].EnthalpyMap_Enthalpy_kJ_kg[8,6] := 498.5881;
   Fluids[2].EnthalpyMap_Enthalpy_kJ_kg[8,7] := 520.3678;
   Fluids[2].EnthalpyMap_Enthalpy_kJ_kg[8,8] := 551.7377;
   Fluids[2].EnthalpyMap_Enthalpy_kJ_kg[9,0] := 397.8677;
   Fluids[2].EnthalpyMap_Enthalpy_kJ_kg[9,1] := 425.8558;
   Fluids[2].EnthalpyMap_Enthalpy_kJ_kg[9,2] := 438.3909;
   Fluids[2].EnthalpyMap_Enthalpy_kJ_kg[9,3] := 462.7447;
   Fluids[2].EnthalpyMap_Enthalpy_kJ_kg[9,4] := 463.5576;
   Fluids[2].EnthalpyMap_Enthalpy_kJ_kg[9,5] := 484.1742;
   Fluids[2].EnthalpyMap_Enthalpy_kJ_kg[9,6] := 497.9508;
   Fluids[2].EnthalpyMap_Enthalpy_kJ_kg[9,7] := 522.3931;
   Fluids[2].EnthalpyMap_Enthalpy_kJ_kg[9,8] := 555.3659;
   Fluids[2].EnthalpyMap_Enthalpy_kJ_kg[10,0] := 403.7939;
   Fluids[2].EnthalpyMap_Enthalpy_kJ_kg[10,1] := 433.1682;
   Fluids[2].EnthalpyMap_Enthalpy_kJ_kg[10,2] := 448.1372;
   Fluids[2].EnthalpyMap_Enthalpy_kJ_kg[10,3] := 467.0842;
   Fluids[2].EnthalpyMap_Enthalpy_kJ_kg[10,4] := 467.3177;
   Fluids[2].EnthalpyMap_Enthalpy_kJ_kg[10,5] := 483.0886;
   Fluids[2].EnthalpyMap_Enthalpy_kJ_kg[10,6] := 498.0977;
   Fluids[2].EnthalpyMap_Enthalpy_kJ_kg[10,7] := 523.751;
   Fluids[2].EnthalpyMap_Enthalpy_kJ_kg[10,8] := 557.4834;
   Fluids[2].EnthalpyMap_Enthalpy_kJ_kg[11,0] := 406.426;
   Fluids[2].EnthalpyMap_Enthalpy_kJ_kg[11,1] := 436.4671;
   Fluids[2].EnthalpyMap_Enthalpy_kJ_kg[11,2] := 452.4549;
   Fluids[2].EnthalpyMap_Enthalpy_kJ_kg[11,3] := 469.0933;
   Fluids[2].EnthalpyMap_Enthalpy_kJ_kg[11,4] := 469.2745;
   Fluids[2].EnthalpyMap_Enthalpy_kJ_kg[11,5] := 483.1994;
   Fluids[2].EnthalpyMap_Enthalpy_kJ_kg[11,6] := 498.3468;
   Fluids[2].EnthalpyMap_Enthalpy_kJ_kg[11,7] := 524.4174;
   Fluids[2].EnthalpyMap_Enthalpy_kJ_kg[11,8] := 558.4523;
   Fluids[1].Limits.T_HeatSourceTemperature_Max := 65.0;
   Fluids[2].Limits.T_HeatSourceTemperature_Max := 120.0;
   Fluids[1].Limits.T_HeatSourceTemperature_Min := 10.0;
   Fluids[2].Limits.T_HeatSourceTemperature_Min := 55.0;
   Fluids[1].Limits.T_HeatSinkTemperature_Max := 85.0;
   Fluids[2].Limits.T_HeatSinkTemperature_Max := 150.0;
   Fluids[1..2].Limits.T_OilTemperature_Critical := 140.0;
   Fluids[1].Limits.T_OilSuperheat := 12.0;
   Fluids[2].Limits.T_OilSuperheat := 15.0;
   Fluids[1..2].Limits.T_CoolingSetpoint := 0.0;
   Fluids[1].T_AdditionalSuperHeatEvaporator := 0.0;
   Fluids[2].T_AdditionalSuperHeatEvaporator := 8.0;
   Fluids[1].P_CriticalPoint := 3583.9;
   Fluids[2].P_CriticalPoint := 3623.637;
   CompressorTypes[1].CompressorTypeNumber := 1;
   CompressorTypes[2].CompressorTypeNumber := 2;
   CompressorTypes[3].CompressorTypeNumber := 3;
   CompressorTypes[4].CompressorTypeNumber := 4;
   CompressorTypes[1].Limits.p_CrankCase_Max := 1600.0;
   CompressorTypes[1].Limits.p_Oil_Min := 90.0;
   CompressorTypes[1].Limits.n_Compressor_Max := 1200.0;
   CompressorTypes[1].Limits.T_Motor_Max := 90.0;
   CompressorTypes[1].Limits.M_Motor_Limit := 61.4;
   CompressorTypes[1].Limits.T_Inverter_Max := 60.0;
   CompressorTypes[1].Constant.CompressionVolume_L := 16.4;
   CompressorTypes[1].Constant.CompressionLostPerPressureRatio := 1.782;   // Theoretisch eher 4.5
   CompressorTypes[1].Constant.PumpEfficinecy := 72.43;   // Theoretisch eher 95
   // SystemTypes[1] : Alpha-1
   // SystemTypes[2] : Alpha-2
   // SystemTypes[3] : Offenau
   SystemTypes[1].SystemTypeNumber := 1;
   SystemTypes[2].SystemTypeNumber := 2;
   SystemTypes[3].SystemTypeNumber := 3;
   SystemTypes[4].SystemTypeNumber := 4;
   SystemTypes[5].SystemTypeNumber := 5;
   SystemTypes[6].SystemTypeNumber := 6;
   SystemTypes[1..2].Limits.T_SuperHeatCompressorIn_Min := 2.0;
   SystemTypes[4..5].Limits.T_SuperHeatCompressorIn_Min := 2.0;
   SystemTypes[1..2].Limits.T_Housing_Max := 50.0;
   SystemTypes[4].Limits.T_Housing_Max := 55.0;
   SystemTypes[5].Limits.T_Housing_Max := 50.0;
   SystemTypes[1].Limits.T_CoolingCycle_Max := 70.0;
   SystemTypes[2].Limits.T_CoolingCycle_Max := 65.0;
   SystemTypes[4..5].Limits.T_CoolingCycle_Max := 110.0;
   SystemTypes[1].Limits.p_CompressorOut_Max := 2590.0;
   SystemTypes[2].Limits.p_CompressorOut_Max := 2700.0;
   SystemTypes[4].Limits.p_CompressorOut_Max := 2950.0;
   SystemTypes[5].Limits.p_CompressorOut_Max := 3000.0;
   SystemTypes[1].Limits.p_EvaporatorOut_Max := 1450.0;
   SystemTypes[2].Limits.p_EvaporatorOut_Max := 1550.0;
   SystemTypes[4..5].Limits.p_EvaporatorOut_Max := 1100.0;
   SystemTypes[5].Settings.CooliungPump_ReversedPWM := true;
   SystemTypes[4].Settings.MotorCooling_AirFanCooledCycle := true;
   SystemTypes[2].Settings.DoubleExpansionValves := true;
END_DATA_BLOCK
